FUNCTION_BLOCK FB_AxisStatusNC IMPLEMENTS I_AxisStatus
VAR_INPUT
END_VAR
VAR_OUTPUT
END_VAR
VAR
    {attribute 'no_copy'}
    AxisRef : REFERENCE TO AXIS_REF;
    bDone : BOOL;
    bBusy    : BOOL;
END_VAR

THIS^.AxisRef.ReadStatus();

METHOD AxisEnabled : BOOL
// Get a definitive bEnabled reading
CASE THIS^.AxisRef.Status.MotionState OF
    // We are not enabled if there is an issue
    MC_AXISSTATE_UNDEFINED, MC_AXISSTATE_DISABLED, MC_AXISSTATE_ERRORSTOP:
        AxisEnabled := FALSE;
    ELSE
        AxisEnabled := TRUE;
END_CASE
END_METHOD

{warning 'add property implementation'}
PROPERTY AxisError : BOOL
GET
AxisError := THIS^.AxisRef.Status.Error;
END_GET
END_PROPERTY

{warning 'add property implementation'}
PROPERTY AxisErrorID : UDINT
GET
AxisErrorID := THIS^.AxisRef.Status.ErrorID;
END_GET
END_PROPERTY

{warning 'add property implementation'}
PROPERTY AxisID : UDINT
GET
AxisId:=THIS^.AxisRef.NcToPlc.AxisId;
END_GET
END_PROPERTY

{warning 'add property implementation'}
PROPERTY AxisState : Tc2_MC2.MC_AxisStates
GET
AxisState := THIS^.AxisRef.Status.MotionState;
END_GET
END_PROPERTY

//FB_Init is always available implicitly and it is used primarily for initialization.
//The return value is not evaluated. For a specific influence, you can also declare the
//methods explicitly and provide additional code there with the standard initialization
//code. You can evaluate the return value.
METHOD FB_Init: BOOL
VAR_INPUT
    bInitRetains: BOOL; // TRUE: the retain variables are initialized (reset warm / reset cold)
    bInCopyCode: BOOL;  // TRUE: the instance will be copied to the copy code afterward (online change)
    AxisRef : REFERENCE TO AXIS_REF;
END_VAR
THIS^.AxisRef REF= AxisRef;
END_METHOD

{warning 'add property implementation'}
PROPERTY InTargetPosition : BOOL
GET
InTargetPosition := THIS^.AxisRef.Status.InTargetPosition;
END_GET
END_PROPERTY

{warning 'add property implementation'}
PROPERTY MeasuredAcceleration : LREAL
GET
MeasuredAcceleration := THIS^.AxisRef.NcToPlc.ActAcc;
END_GET
END_PROPERTY

{warning 'add property implementation'}
PROPERTY MeasuredPosition : LREAL
GET
// (*Actual Position*)
MeasuredPosition:=THIS^.AxisRef.NcToPlc.ActPos;
END_GET
END_PROPERTY

{warning 'add property implementation'}
PROPERTY MeasuredPositionDiff : LREAL
GET
// (*Actual Position Diff*)
MeasuredPositionDiff:=THIS^.AxisRef.NcToPlc.PosDiff;
END_GET
END_PROPERTY

{warning 'add property implementation'}
PROPERTY MeasuredVelocity : LREAL
GET
// (*Actual Velocity*)
MeasuredVelocity:=THIS^.AxisRef.NcToPlc.ActVelo;
END_GET
END_PROPERTY

PROPERTY Message : T_MAXSTRING
GET
END_GET
END_PROPERTY

{warning 'add property implementation'}
PROPERTY NegativeMotionIsEnabled : BOOL
GET
NegativeMotionIsEnabled := THIS^.AxisRef.Status.NegativeDirection;
END_GET
END_PROPERTY

{warning 'add property implementation'}
PROPERTY PositiveMotionIsEnabled : BOOL
GET
PositiveMotionIsEnabled := THIS^.AxisRef.Status.PositiveDirection;
END_GET
END_PROPERTY

PROPERTY StandStill : BOOL
GET
StandStill := THIS^.AxisRef.Status.StandStill;
END_GET
END_PROPERTY

{warning 'Add property implementation'}
PROPERTY Stopped : BOOL
GET
Stopped := THIS^.AxisRef.Status.HasBeenStopped;
END_GET
END_PROPERTY

END_FUNCTION_BLOCK

(* stored: Version 1.1.0.1
   POU FB_AxisStatusNC: Id {48b2ca9e-7e0c-4a40-afd9-65beb0d8f7fb}, SpecialFunc None
   Method AxisEnabled: Id {2a14e841-fea3-4b30-9123-2945a0231bb1}
   Property AxisError: Id {548a6916-d1a2-4d00-87ab-a00f5b019e53}
   Get Get: Id {74afa849-d130-475a-8341-04da63542fc9}
   Property AxisErrorID: Id {368d990c-4118-41ef-8dc7-2a94afb0a374}
   Get Get: Id {d4abb0c7-70be-4b55-8227-7b88913acfef}
   Property AxisID: Id {b55ca9d1-a2f2-480e-8cbb-a4c4afcd2415}
   Get Get: Id {690eb4ae-f09b-4d3e-9b07-69bd8cd447b8}
   Property AxisState: Id {4fd0f177-1ed6-45bb-bff4-4341481e5661}
   Get Get: Id {97db2c6e-eff4-4d18-9d44-7ecc59764d3a}
   Method FB_Init: Id {30149fc9-8e6b-4cfe-b3d9-a8df4e5fe0ba}
   Property InTargetPosition: Id {833e02a9-2ab3-4627-b017-70699d164f13}
   Get Get: Id {61009624-f415-45ec-8a11-0cb9f7b4d0aa}
   Property MeasuredAcceleration: Id {4119321c-b4b8-4129-b781-b94c8b154a94}
   Get Get: Id {20862a9b-2723-4b7b-bca0-95d5609f10fe}
   Property MeasuredPosition: Id {754e7b8a-3eae-48a8-96e0-2df6eb19a0af}
   Get Get: Id {741ffe13-80d1-4fb2-909b-14aaf0799800}
   Property MeasuredPositionDiff: Id {17bea7bf-049e-4340-843e-56e70e8380d9}
   Get Get: Id {b3d1805f-9f5c-480e-adf6-246877ce89b9}
   Property MeasuredVelocity: Id {089d6dec-53ad-4749-b018-c05930c304c5}
   Get Get: Id {b2c7b5e2-059e-44db-bbc9-22d66d2ed3b0}
   Property Message: Id {5ab8dd75-11ac-4ef7-9841-ea47e6bb03ef}
   Get Get: Id {1f07d7ce-3842-4eaf-b982-a682ff02bbfa}
   Property NegativeMotionIsEnabled: Id {352ac11a-7d4b-4d2b-b7c7-013ee91633cc}
   Get Get: Id {30804582-e098-4034-970d-6e91990daaf1}
   Property PositiveMotionIsEnabled: Id {4637d8b1-ec1d-4ec0-be60-4008469f6e35}
   Get Get: Id {295be85a-4e0b-4a6e-8b69-28cb34305fc0}
   Property StandStill: Id {f49bd614-c508-4377-a6b7-0f9eab982958}
   Get Get: Id {f3718d17-a0bb-4000-88b4-c7094834adc0}
   Property Stopped: Id {c6375ac0-08b6-4b85-999a-45c5d7a1fa71}
   Get Get: Id {abded25b-8407-4890-9c37-9bccdbf06f91} *)
